FUNCTION TFWorkareaConPacchiComplete : BOOL
VAR_INPUT
	WorkArea : POINTER TO ARRAY [1..MAXAREA] OF TFMachinePalletizer_WorkArea;
	Forming : POINTER TO ARRAY [1..MAXFORMING] OF TFMachinePalletizer_Forming;
	WorkAreaState : POINTER TO ARRAY [1..MAXAREA] OF TFMachinePalletizer_WorkAreaState;
END_VAR
VAR
	wa : INT;
	n : INT;
	i : INT;
	a : INT;
END_VAR

TFWorkareaConPacchiComplete := TRUE; 

FOR wa:=1 TO MAXAREA DO
	IF WorkArea^[wa].Enable = 1 THEN
		(* Verifico se il codice è già stato assegnato *)
		IF (WorkArea^[wa].Code > 0 AND WorkArea^[wa].Typology = TYPOLOGY_PALLET) AND 
		(WorkAreaState^[wa].State < WORKAREA_STATE_OCCUPIED_WORKED AND WorkAreaState^[wa].State > WORKAREA_STATE_FREE_DISABLED) AND 
		(Forming^[WorkAreaState^[wa].F].PackXP[WorkAreaState^[wa].P].Grip <> -1 AND 
		Forming^[WorkAreaState^[wa].F].PackXN[WorkAreaState^[wa].P].Grip <> -1) THEN
			TFWorkareaConPacchiComplete := FALSE; 
			RETURN;
		END_IF
	END_IF
END_FOR

END_FUNCTION

(* stored: Version 1.1.0.1, ProductVersion 3.1.4024.11
   POU TFWorkareaConPacchiComplete: Id {52bb9255-5907-48e8-a9d1-a2f34535c493}, SpecialFunc None *)
